INTERFACE I_ForwardEnumerator EXTENDS I_Enumerator

END_INTERFACE

(* stored: Version 1.1.0.1, ProductVersion 3.1.4024.12
   Itf I_ForwardEnumerator: Id {923f4da7-1aef-4c51-89c6-c0c12e907372} *)
